(* Schneider Machine Expert - Basic project Questao3.2_FelipeV1_20241008, file version 2.9.0.0 *)
(* ProjectInformations: Name=Novo projeto *)

HARDWARE
  Cpu 0: TM221M16R/G
  EthernetConfiguration: NetworkName=M221, IpAllocationMode=FixedAddress, IpAddress=0.0.0.0, SubnetMask=0.0.0.0
  SerialLineConfiguration: Baud=Baud19200, Parity=ParityEven, DataBits=DataBits8, StopBits=StopBits1, PhysicalMedium=PhysicalMediumRs485, TransmissionMode=TransmissionModeModbusRtu, SlaveId=1, Addressing=SlaveAddressing
  MastTask: UsePeriodScanMode=false, PeriodScan=100
  FastTask: Period=255
  CpuBehavior: StartingMode=StartAsPreviousState, AutoSaveRamOnEeprom=true, WatchdogPeriod=250

SYMBOLS  (address, symbol, comment, settings)
  %I0.0       "L1"
  %I0.1       "L2"
  %I0.2       "D1"
  %I0.3       "D2"
  %Q0.1       "R1"
  %Q0.2       "R2"

POU Novo POU
  (* SectionNumber=1 *)

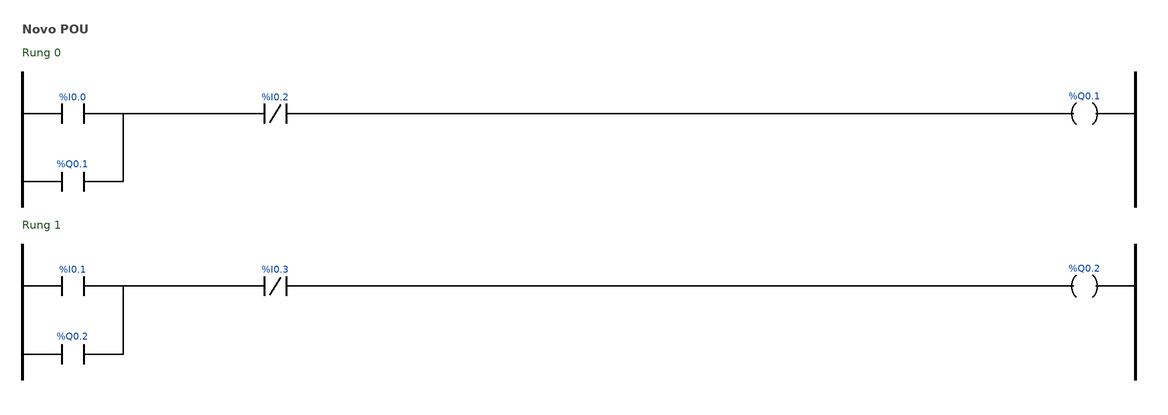

// Rung 0
  LD %I0.0
  OR %Q0.1
  ANDN %I0.2
  ST %Q0.1
  // as ST:
  //   %Q0.1 := (%I0.0 OR %Q0.1) AND NOT %I0.2;

// Rung 1
  LD %I0.1
  OR %Q0.2
  ANDN %I0.3
  ST %Q0.2
  // as ST:
  //   %Q0.2 := (%I0.1 OR %Q0.2) AND NOT %I0.3;
